{attribute addProperty BoxType "EL2521-0000-1022"}
{attribute addProperty Id "StatusAT %I*Status_99BDEBCB1620Counter_valueAT %I*UINT16217"}
{attribute addProperty CRC "2870703641"}
{attribute addProperty SizeInBites "32"}
{attribute addProperty SizeInBytes "4"}
TYPE ENC_Status_compact_AB1B7619 :
STRUCT
	{attribute addProperty Name "Status"}
	Status AT %I* : Status_99BDEBCB;
	{attribute addProperty Name "Counter_value"}
	Counter_value AT %I* : UINT;
END_STRUCT
END_TYPE

(* stored: Version 1.2.0.0, ProductVersion 3.1.4024.9
   DUT ENC_Status_compact_AB1B7619: Id {8bd046cc-1b27-402d-a4fc-0953337ad94a} *)
